FUNCTION_BLOCK ABSTRACT AutomationUnit 
VAR_GENERIC CONSTANT
    _DeviceCount : INT(0..1000) := 0;
END_VAR
EXTENDS Core.Object IMPLEMENTS IAutomationUnit
VAR
	_AutomationRunner : IAutomationRunner;
	
	_LocalSimulationMode : BOOL;	
END_VAR

{attribute 'monitoring' := 'call'}
{attribute 'OPC.UA.DA' := '1'}
{attribute 'OPC.UA.DA.Access' := '1'}
PROPERTY DeviceCount : INT
GET
DeviceCount := _DeviceCount;
END_GET
END_PROPERTY

{attribute 'monitoring' := 'call'}
PROPERTY ABSTRACT Devices : REFERENCE TO ARRAY [0.._DeviceCount - 1] OF Automation.IDevice
GET
END_GET
END_PROPERTY

METHOD FB_init : BOOL
VAR_INPUT
	(* if TRUE, the retain variables are initialized (warm start / cold start)*)
	bInitRetains	: BOOL;
	(* if TRUE, the instance afterwards gets moved into the copy code (online change)*)
	bInCopyCode	: BOOL;
	automationRunner : IAutomationRunner; 
END_VAR
VAR
	automationRunnerNullException : Core.ArgumentNullException;
END_VAR
IF automationRunner = 0 THEN
	automationRunnerNullException.Throw(CurrentNamespace.Name, ClassName, __POUNAME(), __POSITION(), 'automationRunner');
END_IF

_AutomationRunner := automationRunner;
END_METHOD

METHOD FINAL HandleFault
VAR_IN_OUT CONSTANT
	executionContext : AUTOMATION_EXECUTION_CONTEXT;
END_VAR
VAR
	aggregateException : Core.AggregateException;
	
	exceptionCode : __SYSTEM.ExceptionCode;
	exception : IException;
END_VAR
ProcessInputDevices(executionContext, aggregateException);

__TRY
	OnFault(executionContext);
__CATCH(exceptionCode)
	exception := ExceptionManager.GetLastException(exceptionCode);
				
	IF NOT exception.Fatal THEN
		aggregateException.AddInnerException(exception);
	ELSE
		ExceptionManager.ReThrowLastException(exceptionCode);
	END_IF		
__ENDTRY 

ProcessOutputDevices(executionContext, aggregateException);

IF NOT aggregateException.Empty THEN
	aggregateException.Throw(CurrentNamespace.Name, ClassName, __POUNAME(), __POSITION());
END_IF
END_METHOD

METHOD FINAL Initialize : BOOL
VAR_IN_OUT CONSTANT
	executionContext : AUTOMATION_EXECUTION_CONTEXT;
END_VAR
VAR
	i : INT;
		
	exceptionCode : __SYSTEM.ExceptionCode;
	exception : IException;
END_VAR
Initialize := TRUE;

IF __ISVALIDREF(Devices) THEN
	FOR i := 0 TO _DeviceCount - 1 DO
		Initialize := Initialize AND Devices[i].Initialize();
	END_FOR
END_IF

Initialize := Initialize AND OnInitialize();
END_METHOD

{attribute 'monitoring' := 'call'}
{attribute 'OPC.UA.DA' := '1'}
{attribute 'OPC.UA.DA.Access' := '1'}
PROPERTY FINAL LocalSimulationMode : BOOL
GET
LocalSimulationMode := _LocalSimulationMode;
END_GET
END_PROPERTY

METHOD PROTECTED OnFault
VAR_IN_OUT CONSTANT
	executionContext : AUTOMATION_EXECUTION_CONTEXT;
END_VAR
END_METHOD

METHOD PROTECTED OnInitialize : BOOL
OnInitialize := TRUE;
END_METHOD

METHOD PROTECTED ABSTRACT OnRun
VAR_IN_OUT CONSTANT
	executionContext : AUTOMATION_EXECUTION_CONTEXT;
END_VAR
END_METHOD

METHOD PROTECTED OnStop
VAR_IN_OUT CONSTANT
	executionContext : AUTOMATION_EXECUTION_CONTEXT;
END_VAR
END_METHOD

METHOD PRIVATE FINAL processInputDevices
VAR_IN_OUT CONSTANT
	executionContext : AUTOMATION_EXECUTION_CONTEXT;
	aggregateException : Core.AggregateException;
END_VAR
VAR
	i : INT;
	
	inputDevice : IInputDevice;
	
	exceptionCode : __SYSTEM.ExceptionCode;
	exception : IException;
END_VAR
IF NOT __ISVALIDREF(Devices) OR_ELSE _DeviceCount = 0 THEN
	RETURN;
END_IF

FOR i := 0 TO _DeviceCount - 1 DO
	IF NOT __QUERYINTERFACE(Devices[i], inputDevice) THEN
		CONTINUE;
	END_IF
	
	__TRY
		inputDevice.UpdateStateFromInputs(executionContext, aggregateException);
	__CATCH(exceptionCode)
		exception := ExceptionManager.GetLastException(exceptionCode);
					
		IF NOT exception.Fatal THEN
			aggregateException.AddInnerException(exception);
		ELSE
			ExceptionManager.ReThrowLastException(exceptionCode);
		END_IF		
	__ENDTRY 
END_FOR
END_METHOD

METHOD PRIVATE FINAL processOutputDevices
VAR_IN_OUT CONSTANT
	executionContext : AUTOMATION_EXECUTION_CONTEXT;
	aggregateException : Core.AggregateException;
END_VAR
VAR
	i : INT;
	
	outputDevice : IOutputDevice;
	
	exceptionCode : __SYSTEM.ExceptionCode;
	exception : IException;	
END_VAR
IF NOT __ISVALIDREF(Devices) OR_ELSE _DeviceCount = 0 THEN
	RETURN;
END_IF

FOR i := 0 TO _DeviceCount - 1 DO
	IF NOT __QUERYINTERFACE(Devices[i], outputDevice) THEN
		CONTINUE;
	END_IF
	
	__TRY
		outputDevice.UpdateOutputsFromState(executionContext, aggregateException); 
	__CATCH(exceptionCode)
		exception := ExceptionManager.GetLastException(exceptionCode);
					
		IF NOT exception.Fatal THEN
			aggregateException.AddInnerException(exception);
		ELSE
			ExceptionManager.ReThrowLastException(exceptionCode);
		END_IF		
	__ENDTRY 
END_FOR
END_METHOD

METHOD FINAL Run
VAR_IN_OUT CONSTANT
	executionContext : AUTOMATION_EXECUTION_CONTEXT;
END_VAR
VAR
	aggregateException : Core.AggregateException;
	
	exceptionCode : __SYSTEM.ExceptionCode;
	exception : IException;
END_VAR
ProcessInputDevices(executionContext, aggregateException);

__TRY
	OnRun(executionContext);
__CATCH(exceptionCode)
	exception := ExceptionManager.GetLastException(exceptionCode);
				
	IF NOT exception.Fatal THEN
		aggregateException.AddInnerException(exception);
	ELSE
		ExceptionManager.ReThrowLastException(exceptionCode);
	END_IF		
__ENDTRY 

ProcessOutputDevices(executionContext, aggregateException);

IF NOT aggregateException.Empty THEN
	aggregateException.Throw(CurrentNamespace.Name, ClassName, __POUNAME(), __POSITION());
END_IF
END_METHOD

{attribute 'monitoring' := 'call'}
{attribute 'OPC.UA.DA' := '1'}
{attribute 'OPC.UA.DA.Access' := '1'}
PROPERTY FINAL SimulationMode : BOOL
GET
SimulationMode := _LocalSimulationMode OR_ELSE _AutomationRunner.SimulationMode;
END_GET
END_PROPERTY

{attribute 'monitoring' := 'call'}
PROPERTY ABSTRACT StartRequest : BOOL
GET
END_GET
END_PROPERTY

METHOD FINAL Stop
VAR_IN_OUT CONSTANT
	executionContext : AUTOMATION_EXECUTION_CONTEXT;
END_VAR
VAR
	aggregateException : Core.AggregateException;
	
	exceptionCode : __SYSTEM.ExceptionCode;
	exception : IException;
END_VAR
ProcessInputDevices(executionContext, aggregateException);

__TRY
	OnStop(executionContext);
__CATCH(exceptionCode)
	exception := ExceptionManager.GetLastException(exceptionCode);
				
	IF NOT exception.Fatal THEN
		aggregateException.AddInnerException(exception);
	ELSE
		ExceptionManager.ReThrowLastException(exceptionCode);
	END_IF		
__ENDTRY 

ProcessOutputDevices(executionContext, aggregateException);

IF NOT aggregateException.Empty THEN
	aggregateException.Throw(CurrentNamespace.Name, ClassName, __POUNAME(), __POSITION());
END_IF
END_METHOD

{attribute 'monitoring' := 'call'}
PROPERTY StopRequest : BOOL
GET
END_GET
END_PROPERTY

METHOD FINAL TryGetDeviceByIndex : Automation.IDevice
VAR_INPUT
	index : BYTE;
END_VAR
IF index < 0 OR_ELSE index >= _DeviceCount OR_ELSE NOT __ISVALIDREF(Devices) THEN
	RETURN;
END_IF

TryGetDeviceByIndex := Devices[index];
END_METHOD

END_FUNCTION_BLOCK

(* stored: Version 1.1.0.1
   POU AutomationUnit: Id {715bcab9-6d21-43bf-ac33-fb2affdac1da}, SpecialFunc None
   Folder Methods to override: Id {18713aca-9c47-4769-936e-cd3be2ed069c}
   Folder Service memebers: Id {5df4ad11-a7ac-4049-8c04-41c0497c7559}
   Property DeviceCount: Id {612962ce-4a03-4dcb-a1ce-f9e94eefa0eb}
   Get Get: Id {cc518b3a-e440-4848-8075-189e5ee4e093}
   Property Devices: Id {f1c94009-408f-4558-836f-c0ffe07e995d}
   Get Get: Id {3053aa14-2407-42d1-bc4d-bd38e5a9f72c}
   Method FB_init: Id {46ebd59e-7068-435f-99df-fef2ff312630}
   Method HandleFault: Id {5df2316a-8fd1-40c4-8c74-2bd8dd1e2dbf}
   Method Initialize: Id {1b5cfeb5-a4c4-49db-8b34-eb001c2926ca}
   Property LocalSimulationMode: Id {bef27b77-29d7-4729-ae00-5f308c7e5257}
   Get Get: Id {908ef2f4-2445-4cdb-94d6-03aad2842213}
   Method OnFault: Id {47b787a0-74db-428e-a805-17453cf9f9ee}
   Method OnInitialize: Id {f30a4c4a-7966-446f-95b6-a1ce70efb536}
   Method OnRun: Id {f7f57440-8e03-4827-9c8c-4741292bf658}
   Method OnStop: Id {e9a7087e-9b95-447b-8bf1-2d25488d5f40}
   Method processInputDevices: Id {2a706850-e1f1-476b-bd78-85f574de650b}
   Method processOutputDevices: Id {bd8d51f1-abdb-4a43-b7de-c5e6e60ddaf2}
   Method Run: Id {edf960fe-6c94-4ace-a7be-524e71aafd2a}
   Property SimulationMode: Id {d06903e4-ea01-42fc-a468-b432f4fc159b}
   Get Get: Id {c0b7b53d-f5eb-4914-b43e-57840bfbc5da}
   Property StartRequest: Id {efbb592d-bbef-421a-a357-ab7d8e20bcce}
   Get Get: Id {f92effac-0e0d-4aa7-89d3-b6db7e0aeded}
   Method Stop: Id {ef005615-2d66-46a1-8783-315700ef3d6a}
   Property StopRequest: Id {608fa160-a1ee-4b42-a40b-f54246a9eaa1}
   Get Get: Id {ea1fec94-0a94-4c91-97a8-b829d143d2d9}
   Method TryGetDeviceByIndex: Id {822b2535-548b-4af3-814e-271dc3e4c03f} *)
